// TIA Portal project "FactoryIO_Template_S7-1200_V15_V16" (V16)
// Vorlageprojekt für das Buch mit Zielsystem S7-1200

(* hardware
DEVICE "S7-1200-Station_1"  S7-1200 Station
   slot 0: "Baugruppenträger_0"  Rack  V1.0
   slot 1: "PLC_1"  CPU 1211C DC/DC/DC  6ES7 211-1AE40-0XB0  V4.1
*)

// ===== PLC "PLC_1"  CPU 1211C DC/DC/DC =====

VAR_GLOBAL   // PLC tag table "Standard-Variablentabelle"
   "Start" AT %I10.0 : Bool;
   "Stop" AT %I10.1 : Bool;
   "Sensor 1 (Small)" AT %I10.2 : Bool;
   "Sensor 1 (Large)" AT %I10.3 : Bool;
   "Pusher 1 Back Limit(1)" AT %I10.4 : Bool;
   "Pusher 1 Front Limit(1)" AT %I10.5 : Bool;
   "X1" AT %M1.1 : Bool;
   "X2" AT %M1.2 : Bool;
   "Conveyor" AT %Q10.0 : Bool;
   "Pusher 1" AT %Q10.1 : Bool;
   "M" AT %M1.0 : Bool;
   "X3" AT %M1.3 : Bool;
   "X4" AT %M1.4 : Bool;
END_VAR

// folder: System blocks/Program resources

DATA_BLOCK "T1"   // DB1
{ S7_Optimized_Access := 'TRUE' }
AUTHOR : Simatic
FAMILY : IEC
NAME : IEC_TMR
VERSION : 1.0
// stored: InstanceOfName IEC_TIMER
"IEC_TIMER"
BEGIN
END_DATA_BLOCK

// folder: (top level)

FUNCTION "MHJ-PLC-Lab-Function-S71200" : Void   // FC9000, SCL
{ S7_Optimized_Access := 'TRUE' }
VERSION : 0.1
   VAR_TEMP
      rdTimeReturn : Int;
      outputTime : DTL;
      SyncVal : Byte;
      forVal : Int;
      forVal_2 : Int;
      Value : Byte;
   END_VAR
   VAR CONSTANT
      CompVal : Byte := 16#34;
      Value_01 : Byte := 16#11;
      Value_01_DW : DWord := 16#A165_D992;
      Value_02_DW : DWord := 16#58BE_4401;
   END_VAR
BEGIN

   #Value:=PEEK(area := 16#82,
        dbNumber := 0,
        byteOffset := 511);
   #Value := #Value + 1;

   POKE(area := 16#82,
        dbNumber := 0,
        byteOffset := 511,
        value := #Value);

   POKE(area:=16#81,
        dbNumber:=0,
        byteOffset:=1016,
        value:=#Value_01_DW);
   POKE(area := 16#81,
        dbNumber := 0,
        byteOffset := 1020,
        value := #Value_02_DW);

   POKE(area := 16#81,
        dbNumber := 0,
        byteOffset := 511,
        value := B#16#00);

   FOR #forVal := 0 TO 120 DO
       FOR #forVal_2:=0 TO 10 DO
           #rdTimeReturn:=RD_SYS_T(#outputTime);
           #rdTimeReturn := WR_SYS_T(#outputTime);
           #rdTimeReturn := RD_SYS_T(#outputTime);
           #rdTimeReturn := WR_SYS_T(#outputTime);
       END_FOR;
       #SyncVal:= PEEK(area := 16#81,
                      dbNumber := 0,
                      byteOffset := 511);
       IF #SyncVal = #CompVal THEN
          GOTO M_1;
       END_IF;
   END_FOR;
   RETURN;

   M_1:
   POKE(area := 16#81,
        dbNumber := 0,
        byteOffset := 511,
        value := B#16#0);
END_FUNCTION

ORGANIZATION_BLOCK "Main"   // OB1, LAD, ProgramCycle
TITLE = "Main Program Sweep (Cycle)"
{ S7_Optimized_Access := 'TRUE' }
VERSION : 0.1
   VAR_INPUT
      Initial_Call : Bool;   // Initial call of this OB
      Remanence : Bool;   // =True, if remanent data are available
   END_VAR
BEGIN

REGION Network 1: Konnektierungsbaustein für PLC-Lab
   // Im Netzwerk 1 wird der Konnektierungsbaustein für PLC-Lab aufgerufen.
   // Dieser Aufruf darf nicht entfernt werden!
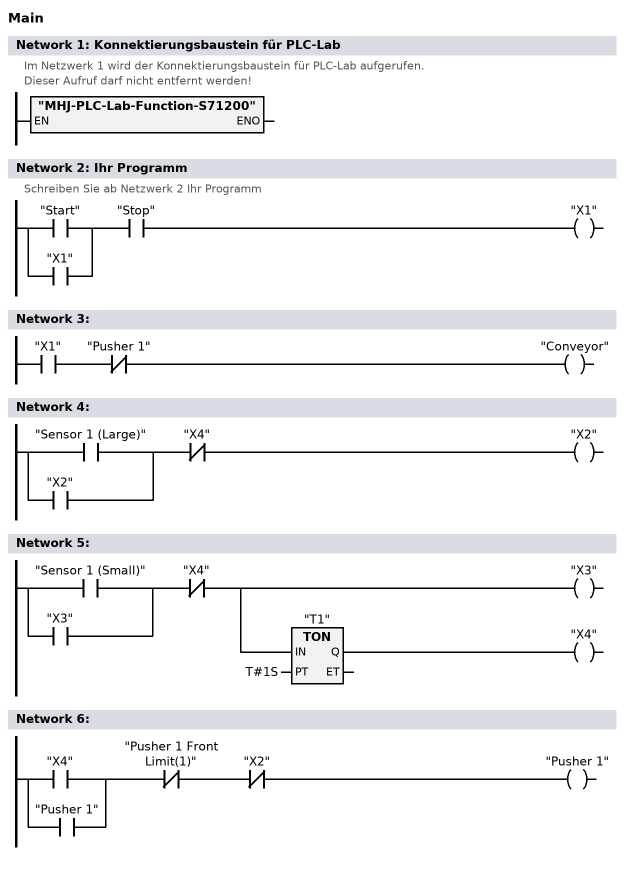
   RUNG wire#powerrail
      "MHJ-PLC-Lab-Function-S71200"()
   END_RUNG
   // the same network as SCL:
   "MHJ-PLC-Lab-Function-S71200"();
END_REGION

REGION Network 2: Ihr Programm
   // Schreiben Sie ab Netzwerk 2 Ihr Programm
   RUNG wire#powerrail
      Contact( "Start" )
      wire#w1
      Contact( "Stop" )
      Coil( "X1" )
   END_RUNG
   RUNG wire#powerrail
      Contact( "X1" )
   END_RUNG wire#w1
   // the same network as SCL:
   "X1" := ("Start" OR "X1") AND "Stop";
END_REGION

REGION Network 3
   RUNG wire#powerrail
      Contact( "X1" )
      I_Contact( "Pusher 1" )
      Coil( "Conveyor" )
   END_RUNG
   // the same network as SCL:
   "Conveyor" := "X1" AND NOT "Pusher 1";
END_REGION

REGION Network 4
   RUNG wire#powerrail
      Contact( "Sensor 1 (Large)" )
      wire#w1
      I_Contact( "X4" )
      Coil( "X2" )
   END_RUNG
   RUNG wire#powerrail
      Contact( "X2" )
   END_RUNG wire#w1
   // the same network as SCL:
   "X2" := ("Sensor 1 (Large)" OR "X2") AND NOT "X4";
END_REGION

REGION Network 5
   "X3" := ("Sensor 1 (Small)" OR "X3") AND NOT "X4";
   "T1".TON(IN := "X3", PT := T#1S);
   "X4" := "T1".Q;
END_REGION

REGION Network 6
   RUNG wire#powerrail
      Contact( "X4" )
      wire#w1
      I_Contact( "Pusher 1 Front Limit(1)" )
      I_Contact( "X2" )
      Coil( "Pusher 1" )
   END_RUNG
   RUNG wire#powerrail
      Contact( "Pusher 1" )
   END_RUNG wire#w1
   // the same network as SCL:
   "Pusher 1" := ("X4" OR "Pusher 1") AND NOT "Pusher 1 Front Limit(1)" AND NOT "X2";
END_REGION
END_ORGANIZATION_BLOCK